// TIA Portal V17 export
// export: Created 2022-07-20T07:01:30.1870398Z, ExportSetting WithDefaults, DisplayName Totally Integrated Automation Portal, DisplayVersion V17, DisplayName TIA Portal Openness, DisplayVersion V17, DisplayName TIA Portal Version Control Interface, DisplayVersion V17, DisplayName SINAMICS Startdrive Advanced, DisplayVersion V17, DisplayName SINAMICS Startdrive G130, G150, S120, S150, SINAMICS MV, S210, DisplayVersion V17, DisplayName SINAMICS Startdrive G110M, G120, G120C, G120D, G120P, G115D, DisplayVersion V17, DisplayName STEP 7 Professional, DisplayVersion V17, DisplayName STEP 7 Safety, DisplayVersion V17, DisplayName WinCC Advanced, DisplayVersion V17
FUNCTION_BLOCK "FB10280_iFoil_L_Control"   // FB10280, LAD
{ S7_Optimized_Access := 'TRUE' }
VERSION : 0.1
// stored: AutoNumber false, IsIECCheckEnabled false, IsRetainMemResEnabled false, MemoryReserve 100, SetENOAutomatically false, UDAEnableTagReadback false
   VAR_INPUT
      iFoilLCommunicationIn : "stiFoilLControlCommunicationIn";
      RequestStartiFoil : Bool;
      RequestStopIFoil : Bool;
   END_VAR
   VAR_OUTPUT
      iFoilLCommunicationOut : "stiFoilLControlCommunicationOut";
      iFoilReady : Bool;
      Standstill : Bool;
      Active : Bool;
      Warning : Bool;
      State_Error : Bool;
   END_VAR
   VAR_IN_OUT
      RequestAcknowledge : Bool;
   END_VAR
   VAR
      R_TRIG_RequestStartiFoil : R_TRIG;
      R_TRIG_RequestStopIFoil { S7_SetPoint := 'True'} : R_TRIG;
      R_TRIG_ResetButton { S7_SetPoint := 'True'} : R_TRIG;
      F_TRIG_RequestStartiFoil : F_TRIG;
      F_TRIG_RequestStopIFoil { S7_SetPoint := 'True'} : F_TRIG;
      F_TRIG_ResetButton { S7_SetPoint := 'True'} : F_TRIG;
      TON_ReadySignalDuration { S7_SetPoint := 'True'} : TON_TIME;
      TON_NotReadySignalDuration { S7_SetPoint := 'True'} : TON_TIME;
      TON_StopSignalDuration { S7_SetPoint := 'True'} : TON_TIME;
   END_VAR
BEGIN

REGION Network 1 (SCL): First Scan
   IF "FirstScan" THEN
       #iFoilReady := FALSE;
       #iFoilLCommunicationOut.DoWarmingUp := FALSE;
       #iFoilLCommunicationOut.DoStop := FALSE;
   END_IF;
END_REGION

REGION Network 2 (SCL): Edge Signals & Timers
   REGION EDGE SIGNALS
       #R_TRIG_RequestStartiFoil(CLK := #RequestStartiFoil);
       #R_TRIG_RequestStopIFoil(CLK := #RequestStopIFoil);

       #F_TRIG_RequestStartiFoil(CLK := #RequestStartiFoil);
       #F_TRIG_RequestStopIFoil(CLK := #RequestStopIFoil);
   END_REGION

   REGION TIMERS
       #TON_ReadySignalDuration(IN := #iFoilLCommunicationIn.Ready,
                                PT := T#3s);

       #TON_NotReadySignalDuration(IN := NOT(#iFoilLCommunicationIn.Ready),
                                PT := T#3s);

       #TON_StopSignalDuration(IN := #RequestStopIFoil AND #iFoilLCommunicationOut.DoStop,
                               PT := T#2s);
   END_REGION
END_REGION

REGION Network 3 (SCL): iFoil Commands Management
   IF #R_TRIG_RequestStartiFoil.Q THEN
       #iFoilLCommunicationOut.DoWarmingUp := TRUE;
       #iFoilLCommunicationOut.DoStop := FALSE;
   ELSIF #R_TRIG_RequestStopIFoil.Q THEN
       #iFoilLCommunicationOut.DoWarmingUp := FALSE;
       #iFoilLCommunicationOut.DoStop := TRUE;
   ELSIF #F_TRIG_RequestStartiFoil.Q OR #F_TRIG_RequestStopIFoil.Q THEN
       #iFoilLCommunicationOut.DoWarmingUp := FALSE;
       #iFoilLCommunicationOut.DoStop := FALSE;
   END_IF;

   IF #R_TRIG_ResetButton.Q THEN
       #RequestAcknowledge := TRUE;
   ELSIF #F_TRIG_ResetButton.Q THEN
       #RequestAcknowledge := FALSE;
   END_IF;
END_REGION

REGION Network 4 (SCL): iFoil States Management
   IF #TON_ReadySignalDuration.Q THEN
       #iFoilReady := TRUE;
   ELSIF #TON_NotReadySignalDuration.Q THEN
       #iFoilReady := FALSE;
   END_IF;

   #Standstill := #iFoilLCommunicationIn.iFoilStatus.%X0;
   #Active := #iFoilLCommunicationIn.iFoilStatus.%X1;
   #Warning := #iFoilLCommunicationIn.iFoilStatus.%X2;
   #State_Error := #iFoilLCommunicationIn.Error OR #iFoilLCommunicationIn.iFoilStatus.%X3;
END_REGION
END_FUNCTION_BLOCK
